// Mitsubishi GX Works2 project: 歩進6ステップリラダー風全1bitシフト   PLC: FX3S

PROGRAM MAIN
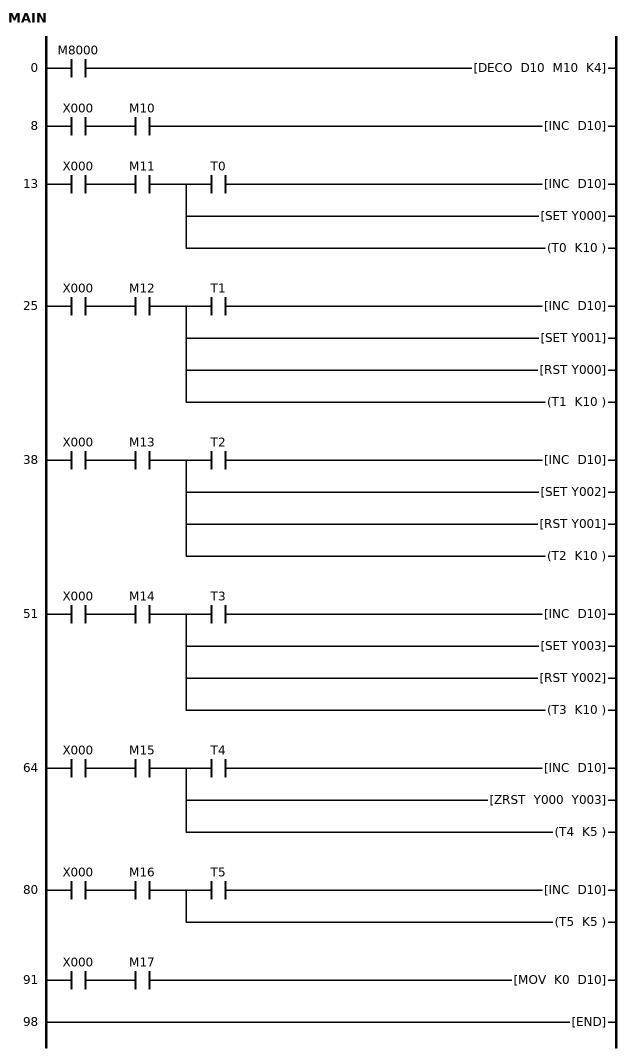
0     LD      M8000
      DECO    D10 M10 K4
8     LD      X000
      AND     M10
      INC     D10
13    LD      X000
      AND     M11
      MPS
      AND     T0
      INC     D10
      MPP
      SET     Y000
      OUT     T0 K10
25    LD      X000
      AND     M12
      MPS
      AND     T1
      INC     D10
      MPP
      SET     Y001
      RST     Y000
      OUT     T1 K10
38    LD      X000
      AND     M13
      MPS
      AND     T2
      INC     D10
      MPP
      SET     Y002
      RST     Y001
      OUT     T2 K10
51    LD      X000
      AND     M14
      MPS
      AND     T3
      INC     D10
      MPP
      SET     Y003
      RST     Y002
      OUT     T3 K10
64    LD      X000
      AND     M15
      MPS
      AND     T4
      INC     D10
      MPP
      ZRST    Y000 Y003
      OUT     T4 K5
80    LD      X000
      AND     M16
      MPS
      AND     T5
      INC     D10
      MPP
      OUT     T5 K5
91    LD      X000
      AND     M17
      MOV     K0 D10
98    END
END_PROGRAM
